TYPE ST_TableControl_HMI :
STRUCT
	iDialogNumber:USINT;
	nCurrentTypeToProduce: nBottleTypes;
	stEditedType:ST_BottleTypeParams;
	nEditedType: nBottleTypes;
	nLastEditedType: nBottleTypes;
	bSave:BOOL;
	bRestore: BOOL;
	bEmptyMode: BOOL;
END_STRUCT
END_TYPE

(* stored: Version 1.1.0.1, ProductVersion 3.1.4024.15
   DUT ST_TableControl_HMI: Id {e9f3e92a-349a-4d66-8583-fd07488f6623} *)
